FUNCTION_BLOCK FB_OPCUA_ClientConnection_Test  EXTENDS TcUnit.FB_TestSuite
VAR_INPUT
END_VAR
VAR_OUTPUT
END_VAR
VAR
END_VAR

errorShouldntBeActiveWhenConnectionIsSuccesful();
errorShouldBeActiveIfConnectingFails();

METHOD errorShouldBeActiveIfConnectingFails
VAR
	connect 				: FB_UAconnectMock_Failure;
	disconnect 				: FB_UAdisconnectMock_success;
	getNameSpaceIndex 		: FB_UAgetNameSpaceIndexMock_success;
	connection 				: FB_OPCUA_ClientConnection(iOPCUAconnect := connect,
														iOPCUAdisconnect := disconnect,
														iOPCUAgetNameSpaceIndex := getNameSpaceIndex);
	sessionCOnnectInfo 		: ST_UASessionConnectInfo;
END_VAR
TEST('errorShouldBeActiveIfConnectingFails');
	connection.connect(serverUrl := '11.11.11.11',
				namespaceUri := 'namespace',
				nameSpaceLocationIdentifier := 'GVL_ident' ,
				sessionConnectInfo := SessionConnectInfo
				);
	assertEquals_BOOL(Expected := TRUE, Actual := connection.error, Message := 'Error not active when connection failed');
TEST_FINISHED();
END_METHOD

METHOD errorShouldntBeActiveWhenConnectionIsSuccesful
VAR
	connect : FB_UAconnectMock_Success;
	disconnect : FB_UAdisconnectMock_success;
	getNameSpaceIndex : FB_UAgetNameSpaceIndexMock_success;
	connection : FB_OPCUA_ClientConnection(iOPCUAconnect := connect,
										iOPCUAdisconnect := disconnect,
										iOPCUAgetNameSpaceIndex := getNameSpaceIndex);
	sessionCOnnectInfo : ST_UASessionConnectInfo;
END_VAR
TEST('errorShouldntBeActiveWhenConnectionIsSuccesful');
	connection.connect(serverUrl := '11.11.11.11',
				namespaceUri := 'namespace',
				nameSpaceLocationIdentifier := 'GVL_ident' ,
				sessionConnectInfo := SessionConnectInfo
				);
	assertEquals_BOOL(Expected := FALSE, Actual := connection.error, Message := 'Error active even when connection succeeced');
TEST_FINISHED();
END_METHOD

END_FUNCTION_BLOCK

(* stored: Version 1.1.0.1, ProductVersion 3.1.4024.9
   POU FB_OPCUA_ClientConnection_Test: Id {7218b254-8f00-48b1-9085-e3c198cc35e1}, SpecialFunc None
   Method errorShouldBeActiveIfConnectingFails: Id {1c941d56-b399-430b-850d-b8e299923506}
   Method errorShouldntBeActiveWhenConnectionIsSuccesful: Id {4f176e35-e4f3-4ca0-9de7-40f0413bc697} *)
